FUNCTION_BLOCK FB_LamparaConmutada_SFC_2
VAR_INPUT
END_VAR
VAR_OUTPUT
END_VAR
VAR
    Lampara AT %Q*: BOOL;
    Pulsador AT %I*: BOOL;
    
    Pulsacion: R_TRIG;
END_VAR

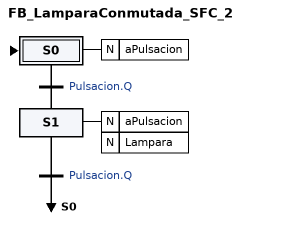
INITIAL_STEP S0:
    aPulsacion(N);
END_STEP
TRANSITION FROM S0 TO S1
    := Pulsacion.Q;
END_TRANSITION
STEP S1:
    aPulsacion(N);
    Lampara(N);
END_STEP
TRANSITION FROM S1 TO S0
    := Pulsacion.Q;
END_TRANSITION

ACTION aPulsacion:
Pulsacion(CLK := Pulsador);
END_ACTION

END_FUNCTION_BLOCK

(* stored: Version 1.1.0.1, ProductVersion 3.1.4024.15
   POU FB_LamparaConmutada_SFC_2: Id {78235adc-5239-4720-b12a-c0069f30d070}, SpecialFunc None
   Action aPulsacion: Id {a2a22992-7e84-4cc8-a09a-7db1500bb18f} *)
